FUNCTION_BLOCK Handling_TeachRack_DlgContent EXTENDS TcoCore.TcoInputDialogContentContainer
VAR
	{attribute addProperty Name "<#Recipe#>"}
	Recipe:STRING;
	{attribute addProperty Name "<#Qantity#>"}
	RequiredQuantity:INT;
	{attribute addProperty Name "<#Timeout#>"}
	Timeout:DATE_AND_TIME;
	{attribute addProperty Name "<#Exclude#>"}
	Exclude:BOOL;
END_VAR

PROPERTY Context : TcoCore.ITcoContext
GET
END_GET
END_PROPERTY

PROPERTY Identity : ULINT
GET
END_GET
END_PROPERTY

END_FUNCTION_BLOCK

(* stored: Version 1.1.0.1
   POU Handling_TeachRack_DlgContent: Id {873ea0b6-a21e-4070-99af-efd2431b7653}, SpecialFunc None
   Property Context: Id {61e85bcd-c4db-4d55-bbd7-3772633141a7}
   Get Get: Id {effd8479-0d8d-4999-9fed-4575de9ba95c}
   Property Identity: Id {f20d0c25-f47e-402a-93af-6534322fc0d6}
   Get Get: Id {cfc99f71-24bf-4def-a38b-ce031ba6e3fb} *)
